Yaskawa INFORM job: R1_W66-67(-70,-90)KM-OK.JBI

/JOB
//NAME R1_W66-67(-70,-90)KM-OK
///FOLDERNAME KRIS-SCIANA
//POS
///NPOS 42,42,0,3,0,0
///TOOL 0
///POSTYPE PULSE
///PULSE
C00000=17054,112532,18066,-13720,97885,70526
C00001=-67216,6920,16605,-16792,61020,-18912
C00002=-106631,-35706,33103,-19473,36985,-59644
C00003=-106518,-29260,43384,-20948,34168,-58800
C00004=-106473,-26428,47849,-21663,32969,-58402
C00005=-106579,-23648,51567,-22137,32148,-58180
C00006=-106473,-26428,47849,-21663,32969,-58402
C00007=-105864,-28760,47081,-22230,32410,-57928
C00008=-105500,-29443,47443,-22664,31948,-57595
C00009=-105864,-28760,47081,-22230,32410,-57928
C00010=-108517,-26795,48156,-21370,32231,-59135
C00011=-110420,-27016,48038,-20892,31842,-59922
C00012=-108517,-26795,48156,-21370,32231,-59135
C00013=-108559,-29650,43668,-20643,33436,-59534
C00014=-108662,-36145,33339,-19149,36264,-60378
C00015=-95607,-50926,18365,20762,46931,-66228
C00016=-91896,-46608,25739,21422,44022,-65495
C00017=-90383,-44735,28852,21715,42833,-65206
C00018=-90835,-41175,33299,22103,42079,-65585
C00019=-90383,-44735,28852,21715,42833,-65206
C00020=-116798,-4764,73813,33023,68695,-35591
C00021=-116763,-2654,77547,33290,67662,-35906
C00022=-116711,-1564,76770,33095,68524,-35620
C00023=-111434,-28935,46331,35007,55009,-71549
C00024=-109336,-28719,46442,35465,54423,-71028
C00025=-111434,-28935,46331,35007,55009,-71549
C00026=-113146,-30211,43694,34249,56316,-71666
C00027=-117250,-32973,37550,32528,59505,-71992
C00028=-93811,55000,78181,-12170,88753,-76596
C00029=-93820,38949,44331,-12503,101061,-77826
C00030=-80223,17432,24206,-5626,82982,-64655
C00031=-82009,-17454,15689,-9029,103119,-33424
C00032=-94073,57506,80607,-12241,88516,-76658
C00033=-93951,54690,76552,-12211,89559,-76721
C00034=-100928,-41248,-5268,10865,87726,-44173
C00035=-63547,-6887,19001,18094,83848,-32102
C00036=-63198,-7482,19877,22790,78533,-33612
C00037=-62716,-6598,20579,22834,78426,-33460
C00038=-87295,15171,28504,-3042,83247,-33138
C00039=-83191,9605,11138,8814,79519,-66133
C00040=-83191,5888,-12199,8726,91833,-65273
C00041=-89356,-161459,-131719,8726,23218,-65273
BC00000=139372,70871,1065839
BC00001=222665,75256,1010845
BC00002=261623,77308,985122
BC00003=261623,77308,985122
BC00004=261623,77308,985122
BC00005=261623,77308,985122
BC00006=261623,77308,985122
BC00007=261623,77308,985122
BC00008=261623,77308,985122
BC00009=261623,77308,985122
BC00010=261623,77308,985122
BC00011=261623,77308,985122
BC00012=261623,77308,985122
BC00013=261623,77308,985122
BC00014=261623,77308,985122
BC00015=305047,122356,942088
BC00016=305047,122356,942088
BC00017=305047,122356,942088
BC00018=305047,122356,942088
BC00019=305047,122356,942088
BC00020=305047,122356,942088
BC00021=305047,122356,942088
BC00022=305047,122356,942088
BC00023=305047,122356,942088
BC00024=305047,122356,942088
BC00025=305047,122356,942088
BC00026=305047,122356,942088
BC00027=305047,122356,942088
BC00028=223613,20045,861305
BC00029=223613,20045,753771
BC00030=175303,17505,740396
BC00031=224648,104771,740537
BC00032=219830,13706,726184
BC00033=219830,13706,726184
BC00034=224648,104771,740537
BC00035=224719,104610,740618
BC00036=224719,104610,740618
BC00037=224719,104610,740618
BC00038=273295,17256,784626
BC00039=227904,17505,857455
BC00040=227904,17505,1049283
BC00041=227904,18593,1049283
///POSTYPE BASE
///RECTAN
///RCONF 0,0,0,0,1,0,0,0,0,0,0,0,0,0,0,0,0,0,0,0,0,0,0,0
P00006=2.006,1.622,-0.565,0.0000,0.0000,0.0000
P00021=0.073,2.058,-0.109,0.0000,0.0000,0.0000
P00022=2.006,1.622,-0.565,0.0000,0.0000,0.0000
//INST
///DATE 2025/04/14 13:14
///ATTR SC,RW
///GROUP1 RB1,BS1
NOP
'r1_W66-67(-70,-90)
'Path S838 (for W504)
SFTOF
MOVJ C00000 BC00000 VJ=100.00
MOVJ C00001 BC00001 VJ=100.00
MOVJ C00002 BC00002 VJ=100.00
MOVJ C00003 BC00003 VJ=100.00
MOVL C00004 BC00004 V=60.0
REFP 3 C00005 BC00005
CALL JOB:SEARCH-R1
SET P021 P006
SFTON P021
MOVL C00006 BC00006 V=60.0
MOVL C00007 BC00007 V=60.0
REFP 3 C00008 BC00008
CALL JOB:SEARCH-R1
SET P021 P006
SFTON P021
MOVL C00009 BC00009 V=60.0
MOVL C00010 BC00010 V=60.0
REFP 3 C00011 BC00011
CALL JOB:SEARCH-R1
SET P021 P006
SFTON P021
MOVL C00012 BC00012 V=60.0
MOVL C00013 BC00013 V=100.0
MOVL C00014 BC00014 V=166.7
'Path S839 (for W504)
SFTOF
MOVJ C00015 BC00015 VJ=100.00
MOVJ C00016 BC00016 VJ=100.00
MOVL C00017 BC00017 V=60.0
REFP 3 C00018 BC00018
CALL JOB:SEARCH-R1
SET P022 P006
SFTON P022
MOVL C00019 BC00019 V=60.0
MOVL C00020 BC00020 V=60.0
REFP 3 C00021 BC00021
CALL JOB:SEARCH-R1
SET P022 P006
SFTON P022
MOVL C00022 BC00022 V=60.0
MOVL C00023 BC00023 V=60.0
REFP 3 C00024 BC00024
CALL JOB:SEARCH-R1
SET P022 P006
SFTON P022
MOVL C00025 BC00025 V=60.0
MOVL C00026 BC00026 V=83.3
MOVL C00027 BC00027 V=83.3
'Path W1362
SFTOF
MOVJ C00028 BC00028 VJ=100.00
MOVJ C00029 BC00029 VJ=100.00
MOVJ C00030 BC00030 VJ=100.00
CALL JOB:COFNIJ_DRUT
SFTON P021
MOVL C00031 BC00031 V=100.0 PL=0
REFP 1 C00032 BC00032
REFP 2 C00033 BC00033
MACRO1 MJ#(0) ARGF7
ARCON
MOVL C00034 BC00034 V=11.2
SFTON P022
MOVL C00035 BC00035 V=11.2
MOVL C00036 BC00036 V=11.2
MOVL C00037 BC00037 V=11.2
ARCOF
MOVL C00038 BC00038 V=83.3
MOVL C00039 BC00039 V=333.3
'Path W1363
SFTOF
MOVL C00040 BC00040 V=333.3
MOVL C00041 BC00041 V=416.7
END
